# EPICS substitutions: evrSupport/Db/evr/evrEventXTA_event.substitutions
#==============================================================================
#
# Abs:  EVR Event Records
#
# Name: evrEventAll.substitutions
#
#==============================================================================
#
file evrPatternProc_event.db {
pattern { DEV       }
	{ $(DEVICE) }
}
